PROGRAM MAIN
VAR
END_VAR

END_PROGRAM

(* stored: Version 1.1.0.1
   POU MAIN: Id {1fdb43d3-1cd5-4878-82bb-e9ca2d43cb5a} *)
